(* PLC project Jaguar, OpenPLC Jaguar 1.0, author OpenPLC Lib Writter *)
(* stored: creationDateTime 2023-04-26T04:54:00, modificationDateTime 2023-04-26T04:54:00 *)

(* Configures the analog channel inputs on the Jaguar board. ADC_CH must be beween 0 - 3. ADC_TYPE must be between 0 - 3, where 0 = unipolar 10V, 1 = bipolar 10V, 2 = unipolar 5V, and 3 = bipolar 5V. Upon successfull configuration of the ADC, SUCCESS is set to TRUE. *)
FUNCTION_BLOCK ADC_CONFIG
  VAR_INPUT
    ADC_CH : SINT;  (* ADC_CH *)
    ADC_TYPE : SINT;  (* ADC_TYPE *)
  END_VAR
  VAR
    ADC_CH_LOCAL : SINT;  (* ADC_CH_LOCAL *)
    ADC_TYPE_LOCAL : SINT;  (* ADC_TYPE_LOCAL *)
  END_VAR
  VAR_OUTPUT
    SUCCESS : BOOL;  (* SUCCESS *)
  END_VAR

  IF ADC_CH <> ADC_CH_LOCAL OR ADC_TYPE <> ADC_TYPE_LOCAL THEN
    ADC_CH_LOCAL := ADC_CH;
    ADC_TYPE_LOCAL := ADC_TYPE;
    SUCCESS := TRUE;
  ELSE
    SUCCESS := FALSE;
  END_IF;
END_FUNCTION_BLOCK
